// TwinCAT 3 PLC project PLC
// ProgramVersion: 3.1.4024.0
// libraries:
//   Tc2_Standard, * (Beckhoff Automation GmbH)
//   Tc2_System, * (Beckhoff Automation GmbH)
//   Tc3_Module, * (Beckhoff Automation GmbH)
//   VisuSymbols,3.5.10.0,System
// project tree:
//   / GlobalTextList.TcGTLO, PlcTask.TcTTO, Visualization Manager.TcVMO (not stored), Visualization.TcVIS
//   POUs/ DoorControl.TcPOU, MotorSimulation.TcPOU, MAIN.TcPOU, VisuSim.TcPOU
// real-time tasks:
//   TASK PlcTask: cycle T#10ms, priority 20, ADS port 350

CONFIGURATION PLC
    RESOURCE PLC ON TwinCAT3
        TASK PlcTask(INTERVAL := T#10ms, PRIORITY := 20);
        PROGRAM MAIN WITH PlcTask : MAIN;
    END_RESOURCE
END_CONFIGURATION

// ---- POUs/MAIN.TcPOU
PROGRAM MAIN
VAR
	DoorControl 		: DoorControl;
	Pb01Sim				: MotorSimulation;
	Pb02Sim				: MotorSimulation;
	PbOut1				: BOOL;
	PbIn1				: BOOL;
	PbOut2				: BOOL;
	PbIn2				: BOOL;
	
	LsDoor1Closed		: BOOL;
	LsDoor1Opened		: BOOL;
	LsDoor2Closed		: BOOL;
	LsDoor2Opened		: BOOL;

	MotorDoor01Open		: BOOL;
	MotorDoor01Close	: BOOL;
	MotorDoor02Open		: BOOL;
	MotorDoor02Close	: BOOL;
	CmdOpen				: BOOL;
	CmdClose			: BOOL;
END_VAR


Pb01Sim(CmdOpen := MotorDoor01Open,
		CmdClose := MotorDoor01Close,
		LsDoorClosed => LsDoor1Closed,
		LsDoorOpened => LsDoor1Opened);
		
Pb02Sim(CmdOpen := MotorDoor02Open,
		CmdClose := MotorDoor02Close,
		LsDoorClosed => LsDoor2Closed,
		LsDoorOpened => LsDoor2Opened);

VisuSim();
		
DoorControl(
	PbOut1:= PbOut1, 
	PbIn1:= PbIn1, 
	LsDoor1Closed:= LsDoor1Closed, 
	LsDoor1Opened:= LsDoor1Opened, 
	PbOut2:= PbOut2, 
	PbInt2:= PbIn2, 
	LsDoor2Closed:= LsDoor2Closed, 
	LsDoor2Opened:= LsDoor2Opened, 
	MotorDoor01Open=> MotorDoor01Open, 
	MotorDoor01Close=> MotorDoor01Close, 
	MotorDoor02Open=> MotorDoor02Open, 
	MotorDoor02Close=> MotorDoor02Close);

END_PROGRAM

// ---- POUs/DoorControl.TcPOU
FUNCTION_BLOCK DoorControl
VAR_INPUT
	PbOut1					:	BOOL;		// Pushbutton outside - door 1
	PbIn1					:	BOOL;		// Pushbutton inside - door 1
	LsDoor1Closed			:	BOOL;		// limit switch door 1 closed
	LsDoor1Opened			:	BOOL;		// limit switch door 1 opened
	
	PbOut2					:	BOOL;		// Pushbutton outside - door 2
	PbInt2					:	BOOL;		// Pushbutton inside - door 2
	LsDoor2Closed			:	BOOL;		// limit switch door 2 closed
	LsDoor2Opened			:	BOOL;		// limit switch door 2 opened
END_VAR
VAR_OUTPUT
	MotorDoor01Open			:	BOOL;		// door 1 - motor open command
	MotorDoor01Close		:	BOOL;		// door 1 - motor close command
	MotorDoor02Open			:	BOOL;		// door 2 - motor open command
	MotorDoor02Close		:	BOOL;		// door 2 - motor close command
END_VAR
VAR
	OneShot					: BOOL := TRUE;	// one shot after power recycle

	OpnSingleDoor01			: SR;			// open only door 1 request 		
	OpnDoor01Request		: SR;			// open door 1 request (door 2 following )
	OpnDoor02Request		: SR;			// open door 2 request (door 1 following)
	OpnDoor01RequestMem		: SR;			// open door 1 request memory
	OpnDoor02RequestMem		: SR;			// open door 2 request memory
	
	Wait					: SR;			// state machine: Wait	
	OpenDoor01Cmd			: SR;			// state machine: open door 1 command
	CloseDoor01Cmd			: SR;			// state machine: close door 1 command
	tonCloseDoor01Cmd		: TON;			// delay open door 1 command
	
	OpenDoor02Cmd			: SR;			// state machine: open door 2 command
	CloseDoor02Cmd			: SR;			// state machine: close door 2 command
	tonCloseDoor02Cmd		: TON;			// delay open door 2 command


	Door02Closed			: SR;			// state machine: door 1 closed
	Door01Closed			: SR;			// state machine: door 2 closed			
	
END_VAR

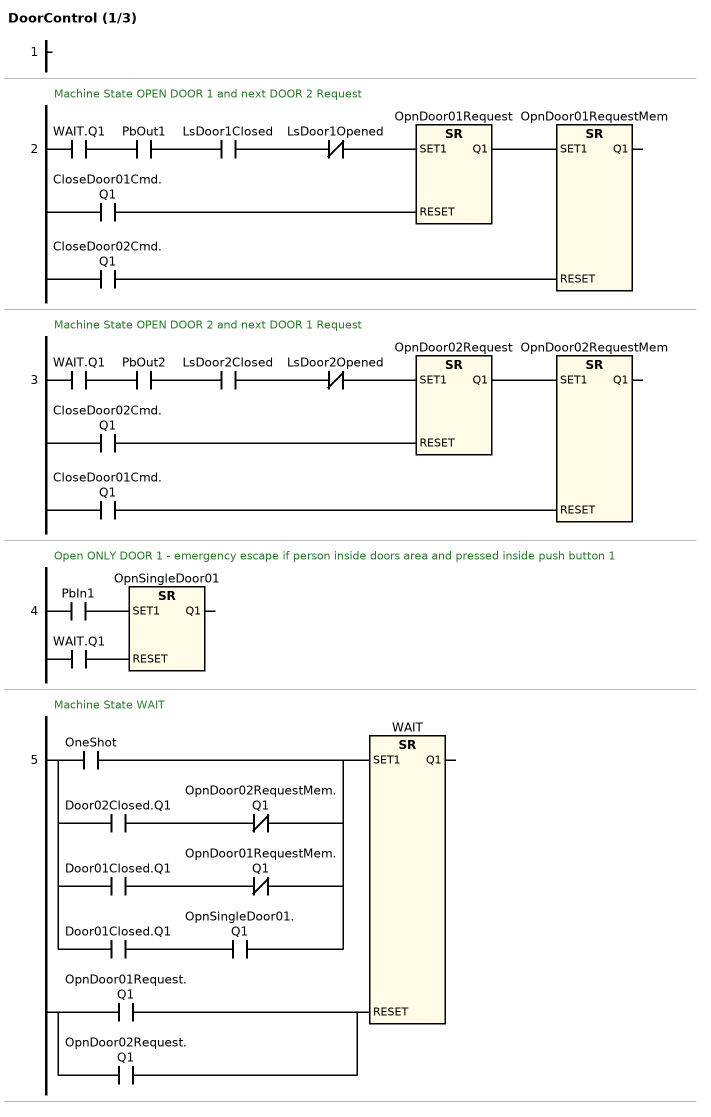
// NETWORK 1

// NETWORK 2
// Machine State OPEN DOOR 1 and next DOOR 2 Request
OpnDoor01Request(SET1 := WAIT.Q1 AND PbOut1 AND LsDoor1Closed AND NOT LsDoor1Opened, RESET := CloseDoor01Cmd.Q1); // SR
OpnDoor01RequestMem(SET1 := OpnDoor01Request.Q1, RESET := CloseDoor02Cmd.Q1); // SR

// NETWORK 3
// Machine State OPEN DOOR 2 and next DOOR 1 Request
OpnDoor02Request(SET1 := WAIT.Q1 AND PbOut2 AND LsDoor2Closed AND NOT LsDoor2Opened, RESET := CloseDoor02Cmd.Q1); // SR
OpnDoor02RequestMem(SET1 := OpnDoor02Request.Q1, RESET := CloseDoor01Cmd.Q1); // SR

// NETWORK 4
// Open ONLY DOOR 1 - emergency escape if person inside doors area and pressed inside push button 1
OpnSingleDoor01(SET1 := PbIn1, RESET := WAIT.Q1); // SR

// NETWORK 5
// Machine State WAIT
WAIT(SET1 := OneShot OR Door02Closed.Q1 AND NOT OpnDoor02RequestMem.Q1 OR Door01Closed.Q1 AND NOT OpnDoor01RequestMem.Q1 OR Door01Closed.Q1 AND OpnSingleDoor01.Q1, RESET := OpnDoor01Request.Q1 OR OpnDoor02Request.Q1); // SR

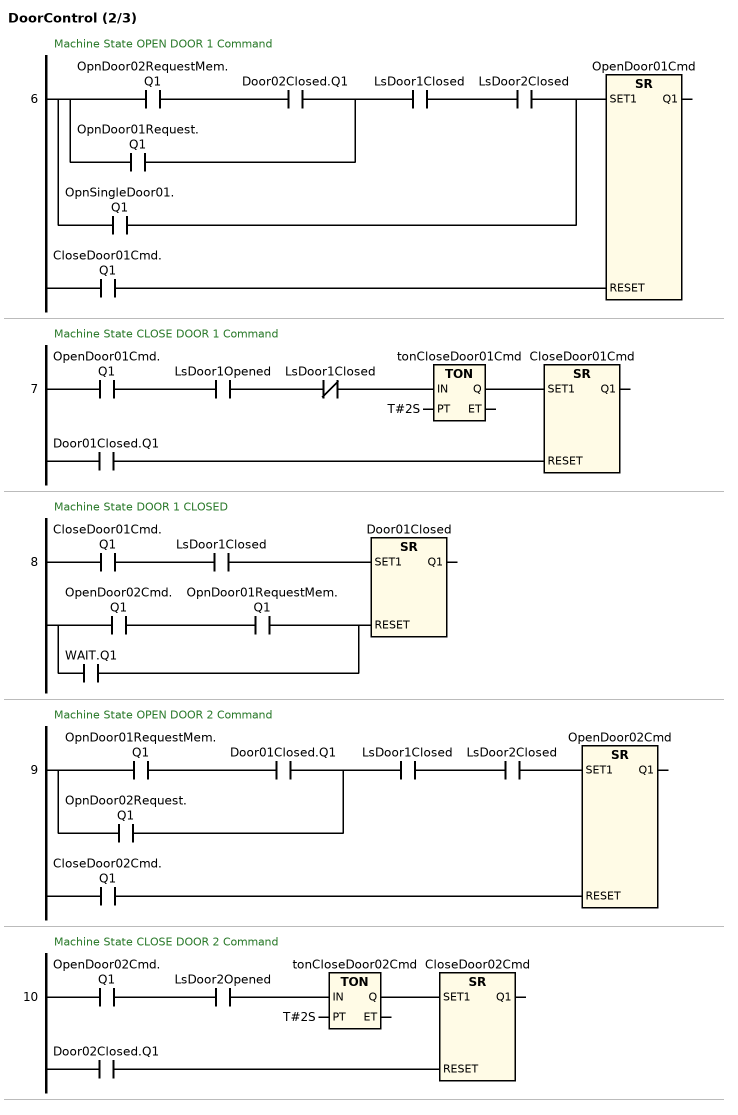
// NETWORK 6
// Machine State OPEN DOOR 1 Command
OpenDoor01Cmd(SET1 := (OpnDoor02RequestMem.Q1 AND Door02Closed.Q1 OR OpnDoor01Request.Q1) AND LsDoor1Closed AND LsDoor2Closed OR OpnSingleDoor01.Q1, RESET := CloseDoor01Cmd.Q1); // SR

// NETWORK 7
// Machine State CLOSE DOOR 1 Command
tonCloseDoor01Cmd(IN := OpenDoor01Cmd.Q1 AND LsDoor1Opened AND NOT LsDoor1Closed, PT := T#2S); // TON
CloseDoor01Cmd(SET1 := tonCloseDoor01Cmd.Q, RESET := Door01Closed.Q1); // SR

// NETWORK 8
// Machine State DOOR 1 CLOSED
Door01Closed(SET1 := CloseDoor01Cmd.Q1 AND LsDoor1Closed, RESET := OpenDoor02Cmd.Q1 AND OpnDoor01RequestMem.Q1 OR WAIT.Q1); // SR

// NETWORK 9
// Machine State OPEN DOOR 2 Command
OpenDoor02Cmd(SET1 := (OpnDoor01RequestMem.Q1 AND Door01Closed.Q1 OR OpnDoor02Request.Q1) AND LsDoor1Closed AND LsDoor2Closed, RESET := CloseDoor02Cmd.Q1); // SR

// NETWORK 10
// Machine State CLOSE DOOR 2 Command
tonCloseDoor02Cmd(IN := OpenDoor02Cmd.Q1 AND LsDoor2Opened, PT := T#2S); // TON
CloseDoor02Cmd(SET1 := tonCloseDoor02Cmd.Q, RESET := Door02Closed.Q1); // SR

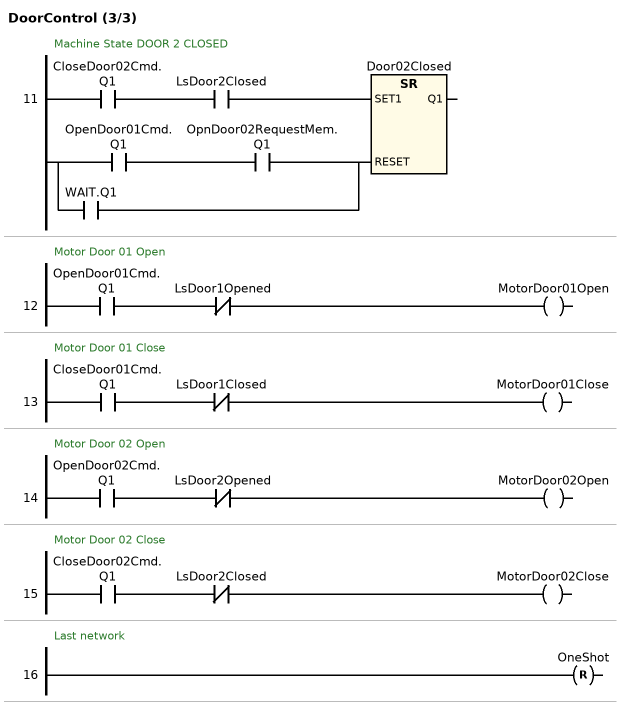
// NETWORK 11
// Machine State DOOR 2 CLOSED
Door02Closed(SET1 := CloseDoor02Cmd.Q1 AND LsDoor2Closed, RESET := OpenDoor01Cmd.Q1 AND OpnDoor02RequestMem.Q1 OR WAIT.Q1); // SR

// NETWORK 12
// Motor Door 01 Open
MotorDoor01Open := OpenDoor01Cmd.Q1 AND NOT LsDoor1Opened;

// NETWORK 13
// Motor Door 01 Close
MotorDoor01Close := CloseDoor01Cmd.Q1 AND NOT LsDoor1Closed;

// NETWORK 14
// Motor Door 02 Open
MotorDoor02Open := OpenDoor02Cmd.Q1 AND NOT LsDoor2Opened;

// NETWORK 15
// Motor Door 02 Close
MotorDoor02Close := CloseDoor02Cmd.Q1 AND NOT LsDoor2Closed;

// NETWORK 16
// Last network
OneShot R= TRUE;

END_FUNCTION_BLOCK

// ---- POUs/MotorSimulation.TcPOU
FUNCTION_BLOCK MotorSimulation
VAR_INPUT
	CmdOpen					:	BOOL;
	CmdClose				:	BOOL;
END_VAR
VAR_OUTPUT
	LsDoorClosed			:	BOOL:=TRUE;
	LSDoorOpened			:	BOOL:=FALSE;
END_VAR
VAR
	tonOpen					:	TON;
	tonClose				:	TON;
END_VAR

IF CmdClose THEN
	tonClose.In:=TRUE;
END_IF

IF CmdOpen THEN
	tonOpen.In:=TRUE;
END_IF

IF tonOpen.Q THEN 
	tonOpen.In:=FALSE;
	LsDoorClosed := FALSE;
	LSDoorOpened := TRUE;
END_IF

IF tonClose.Q THEN 
	tonClose.In:=FALSE;
	LsDoorClosed := TRUE;
	LSDoorOpened := FALSE;
END_IF

tonOpen(PT:=T#1S);
tonClose(PT:=T#1S);

END_FUNCTION_BLOCK

// ---- POUs/VisuSim.TcPOU
PROGRAM VisuSim
VAR
	Door01Pos				:	UINT;
	Door02Pos				:	UINT;
END_VAR

IF MAIN.LsDoor1Opened THEN
	Door01Pos := 120;
ELSIF MAIN.LsDoor1Closed THEN
	Door01Pos := 0;
END_IF


IF MAIN.LsDoor2Opened THEN
	Door02Pos := 120;
ELSIF MAIN.LsDoor2Closed THEN
	Door02Pos := 0;
END_IF

END_PROGRAM

// ---- GlobalTextList.TcGTLO
TEXTLIST GlobalTextList
  226 = 'Door 1'
  853 = 'Door 2'
  864 = 'Door open push b utton'
  744 = 'Door open push button'
  706 = 'Inside Door open PB'
  865 = 'LS\nclosed'
  663 = 'LS\nopened'
  836 = 'M1'
  497 = 'M1\nclose'
  58 = 'M1\nopen'
  479 = 'M2\nclose'
  547 = 'M2\nopen'
END_TEXTLIST

// ---- Visualization.TcVIS
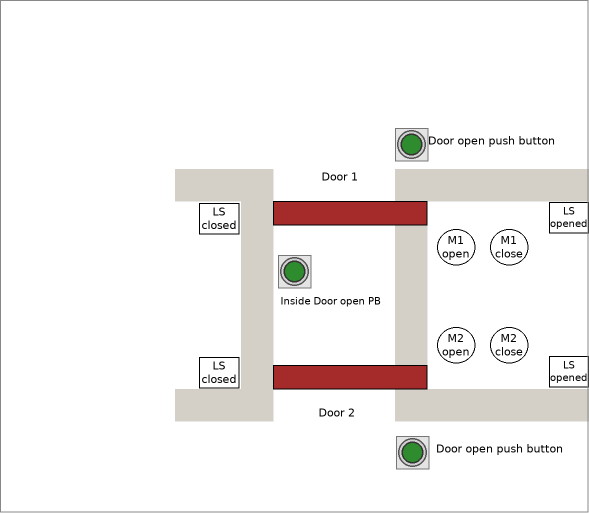
VISUALIZATION Visualization  // 589x513
    Rectangle (241,169 32x252)
    Rectangle (192,152 32x66), angle 90
    Rectangle (192,372 32x66), angle 90
    Rectangle (395,169 32x252)
    Rectangle (519,77 32x216), angle 90
    Rectangle (519,297 32x216), angle 90
    Rectangle (338,136 24x154), angle 90
        p3560616238: VisuSim.Door01Pos
    Rectangle (338,300 24x154), angle 90
        p3560616238: VisuSim.Door02Pos
    Label (309,162 62x30), "Door 1"
    Label (301,398 72x30), "Door 2"
    PushSwitch (395,126 33x37), variable: MAIN.PbOut1, behaviour: TAP, style: Switch-PushSwitch-Green
    PushSwitch (396,434 33x37), variable: MAIN.PbOut2, behaviour: TAP, style: Switch-PushSwitch-Green
    Label (421,126 141x30), "Door open push button"
    Label (429,434 141x30), "Door open push button"
    Ellipse (437,229 38x36), "M1 open", colour toggle: MAIN.MotorDoor01Open
    Ellipse (490,229 38x36), "M1 close", colour toggle: MAIN.MotorDoor01Close
    Ellipse (437,327 38x36), "M2 open", colour toggle: MAIN.MotorDoor02Open
    Ellipse (490,327 38x36), "M2 close", colour toggle: MAIN.MotorDoor02Close
    RoundedRectangle (199,203 40x31), "LS closed", colour toggle: MAIN.LsDoor1Closed
    RoundedRectangle (549,202 40x31), "LS opened", colour toggle: MAIN.LsDoor1Opened
    RoundedRectangle (199,357 40x31), "LS closed", colour toggle: MAIN.LsDoor2Closed
    RoundedRectangle (549,356 40x31), "LS opened", colour toggle: MAIN.LsDoor2Opened
    PushSwitch (278,253 33x37), variable: MAIN.PbIn1, behaviour: TAP, style: Switch-PushSwitch-Green
    Label (271,286 120x30), "Inside Door open PB"
END_VISUALIZATION
